TYPE "Analogic_SensorManagement_Par"
VERSION : 0.1
// Block: Analogic_SensorManagement_Par
   STRUCT
      Enable : Bool;
      RangeLow : Real;
      RangeHigh : Real;
   END_STRUCT;

END_TYPE
